// Annex G worked example on the base class: PLCopen Motion behind the standard
// handshake (S10.6). The parent Unit commands MOVE_TO exactly as it commands a
// cylinder EXTEND - it neither knows nor cares that a servo is involved (S6.1).
//
// The drive is reached ONLY through AXIS_REF and Tc2_MC2. That is what makes the
// type drive-agnostic: a Jenny Science XENAX linked as a CiA402 EtherCAT axis, a
// Beckhoff AX5000, or a simulated NC axis are the same code here. Any
// vendor-specific facility belongs in the driver layer (S10.2), never in a
// reusable CM.
//
// Like FB_SeparatorCM this type declares NO interlocks of its own (S7.2.1). Safe
// motion lives in the certified system; this module only READS its status, and
// the application supplies that status - and any station policy - through
// DeclareCondition/SetCondition. A library cannot name "STO cleared" for a
// station it has never seen.
FUNCTION_BLOCK FB_AxisCM EXTENDS FB_ControlModuleBase
VAR_INPUT
    Command : E_AxisCommand;
    ParCfg : ST_AxisParCfg;
    ParCmd : ST_AxisParCmd;
END_VAR
VAR_OUTPUT
    OutCmd : ST_AxisOutCmd;
    OutImm : ST_AxisOutImm;
    Intlk  : FB_PermIntlk;
END_VAR
VAR CONSTANT
    // §3.8b - the layout version of this module's StationCfg. It belongs with
    // the type that owns the structure, not in the reason band. Bump it when a
    // member is added or its meaning changes (§13).
    AXIS_STATIONCFG_SCHEMA : UINT := 2;   // v2 added JogRequiresEnable
END_VAR
VAR PERSISTENT
    // §3.8b - the retained image. PERSISTENT is the BACKING, not the architecture:
    // the value is registered per (Scope, WriteKey) like every other editable
    // value, so when a set store (file/JSON/XML, MES, asset system) is wired it
    // projects this through the same walk with no change here.
    // Only the VALUE is persistent - the registry's pTarget stays in ordinary
    // VAR, because a retained POINTER names nothing after a restart
    // (ST_ConfigWriteDef, TC3 §3.8b).
    _station : ST_AxisStationCfg;
END_VAR
VAR
    {attribute 'OPC.UA.DA' := '0'}
    _axis : REFERENCE TO AXIS_REF;
    {attribute 'OPC.UA.DA' := '0'}
    _recipe : I_RecipeProvider;
    {attribute 'OPC.UA.DA' := '0'}
    _power : MC_Power;
    {attribute 'OPC.UA.DA' := '0'}
    _homeFb : MC_Home;
    {attribute 'OPC.UA.DA' := '0'}
    _moveFb : MC_MoveAbsolute;
    {attribute 'OPC.UA.DA' := '0'}
    _stopFb : MC_Stop;
    {attribute 'OPC.UA.DA' := '0'}
    _resetFb : MC_Reset;
    {attribute 'OPC.UA.DA' := '0'}
    _jogFb : MC_Jog;
    _jogSeen   : BOOL;   // a held request arrived THIS scan (freshness, O10)
    _jogReqDir : INT;    // +1 / -1 / 0 as last asked
    _jogEnabled: BOOL;   // an enabling device was held when it was asked
    _jogDriving: BOOL;   // the axis is being jogged right now
    _tJogStale : TON;
    _tMove : TON;
    _homed : BOOL;
    _parCfgStaged : ST_AxisParCfg;
    _recipePrepared : BOOL;
    _appCond : ARRAY[1..PL_Fraktal.MAX_PERMINTLK_COND] OF BOOL;
END_VAR

Cyclic();

METHOD PROTECTED OnCyclic : DINT
OnCyclic := SUPER^.OnCyclic();
_M_ApplyConditions();
Intlk();
IF __ISVALIDREF(_axis) THEN                  // defensive (S5.6) [TC3]
    // Enable follows the declared conditions. Losing one drops the enable in the
    // same scan it is lost; re-enabling after it returns is a deliberate command,
    // never automatic (S9.3, S9.4).
    _power(Axis := _axis, Enable := Intlk.AllOk, Enable_Positive := Intlk.AllOk,
        Enable_Negative := Intlk.AllOk, Override := 100.0);
    OutImm.ActPos := _axis.NcToPlc.ActPos;
    OutImm.ActVelocity := _axis.NcToPlc.ActVelo;
    OutImm.DriveEnabled := _power.Status;
END_IF
_M_JogCyclic();
OutImm.TaughtPosition := _station.TaughtPosition;
OutImm.Homed := _homed;
OutCmd.Homed := _homed;
OutImm.Diagnostic := Status.Diagnostic;
END_METHOD

METHOD PRIVATE _M_ApplyConditions
VAR
    i : INT;
END_VAR
FOR i := 1 TO PL_Fraktal.MAX_PERMINTLK_COND DO
    Intlk.Cond[i] := _appCond[i];
END_FOR
END_METHOD

// Core S7.2.1 - the application names its own conditions on this module; the
// library declares none. Safe-motion status (S9.2) is read-only application
// input, so "STO cleared" is declared here by the station that can see it.
// Declared conditions start FALSE: declaring one states an intent to gate.
METHOD DeclareCondition : BOOL
VAR_INPUT
    Index : INT;
    DescriptionKey : STRING(255);
    Reason : E_Reason;
    Bypassable : BOOL;
END_VAR
IF (Index < 1) OR (Index > PL_Fraktal.MAX_PERMINTLK_COND) THEN
    DeclareCondition := FALSE;
    RETURN;
END_IF
_appCond[Index] := FALSE;
DeclareCondition := Intlk.Define(Index := Index, Description := DescriptionKey,
    Reason := Reason, Bypassable := Bypassable);
END_METHOD

// Drive a condition declared by DeclareCondition, every scan.
METHOD SetCondition : BOOL
VAR_INPUT
    Index : INT;
    Ok : BOOL;
END_VAR
IF (Index < 1) OR (Index > PL_Fraktal.MAX_PERMINTLK_COND) THEN
    SetCondition := FALSE;
    RETURN;
END_IF
_appCond[Index] := Ok;
SetCondition := TRUE;
END_METHOD

// §7.6.1 held command - JOG_POS / JOG_NEG. Called EVERY SCAN while the
// operator holds the button; silence stops the axis (see _M_JogCyclic).
//
// This method only RECORDS the request. Nothing moves from here: the decision to
// drive is taken once per scan in _M_JogCyclic, where the interlock, the enabling
// device, the freshness deadline and the command handshake are all weighed
// together. Keeping the decision in one place is what makes it reviewable.
METHOD RequestHeldCommand : BOOL
VAR_INPUT
    Value  : DINT;
    Enable : ST_ManualEnableStatus;
END_VAR
// IF rather than CASE: a CASE label must be a compile-time constant, and
// TO_DINT(enum) is a call. The intent is the same - a defined ELSE (§5.6).
IF Value = TO_DINT(E_AxisCommand.JOG_POS) THEN
    _jogReqDir :=  1;
ELSIF Value = TO_DINT(E_AxisCommand.JOG_NEG) THEN
    _jogReqDir := -1;
ELSE
    // Not a held command of this type. Refuse, and do not record it - an unknown
    // value must never leave a stale direction behind.
    RequestHeldCommand := FALSE;
    RETURN;
END_IF

_jogSeen    := TRUE;
_jogEnabled := Enable.Held;

// Refused up front, with the reason, when no safety-rated enabling device is
// permitting. The axis ALSO has to pass its interlocks in _M_JogCyclic - this is
// an additional requirement, never a way around them (§9).
//
// StationCfg.JogRequiresEnable is what an installation WITHOUT an enabling
// device declares (§3.8a). It relaxes exactly this one requirement: the
// interlocks, the freshness deadline and the command handshake are untouched,
// so a station that declares it still cannot jog through a dropped interlock
// or on a stale request.
IF _station.JogRequiresEnable AND NOT Enable.Held THEN
    OutImm.JogStopReason := PL_ModuleReasons.AXIS_JOG_NOT_ENABLED;
    RequestHeldCommand := FALSE;
    RETURN;
END_IF
RequestHeldCommand := TRUE;
END_METHOD

// The one place a jog is allowed to start, continue, or stop. Runs every scan
// from OnCyclic, whether or not anybody asked - because "nobody asked" is
// precisely the condition that has to stop the axis.
METHOD PRIVATE _M_JogCyclic
VAR
    drive : BOOL;
END_VAR
// Freshness (O10). The timer accumulates while no request arrives, so a caller
// that goes quiet - operator released, HMI closed, network stalled with the
// button still down - stops the axis after JogTimeout. A few scans of jitter are
// tolerated; a dead transport is not.
_tJogStale(IN := NOT _jogSeen, PT := ParCfg.JogTimeout);

// Every gate that must hold for the axis to move by hand, in one expression so
// there is one place to review. Interlocks are NOT bypassed for teaching: the
// station is expected to have wired its guard condition so the safety system's
// teach grant satisfies it, and if it has not, the axis simply does not jog
// (§7.2.1, fail-closed).
drive := (_jogReqDir <> 0)
    AND NOT _tJogStale.Q
    AND (_jogEnabled OR NOT _station.JogRequiresEnable)
    AND Intlk.AllOk
    AND NOT Busy                        // a commanded move owns the axis (§6.1)
    AND __ISVALIDREF(_axis);

// Say why it stopped, once, on the transition. Published status, not an alarm.
IF _jogDriving AND NOT drive THEN
    // The PLC genuinely cannot tell "operator let go" from "link died" - both
    // are simply the request no longer arriving - so it reports what it knows
    // rather than inventing a distinction. The HMI CAN tell, because it knows
    // whether it is still sending, and surfaces the difference there.
    IF _tJogStale.Q THEN
        OutImm.JogStopReason := PL_ModuleReasons.AXIS_JOG_RELEASED;
    ELSIF NOT _jogEnabled AND _station.JogRequiresEnable THEN
        OutImm.JogStopReason := PL_ModuleReasons.AXIS_JOG_NOT_ENABLED;
    ELSIF NOT Intlk.AllOk THEN
        OutImm.JogStopReason := TO_DINT(E_Reason.INTERLOCK_DROPPED);
    ELSE
        OutImm.JogStopReason := PL_ModuleReasons.AXIS_JOG_RELEASED;
    END_IF
    _jogReqDir := 0;
END_IF

IF __ISVALIDREF(_axis) THEN
    _jogFb(Axis := _axis,
           JogForward   := drive AND (_jogReqDir > 0),
           JogBackwards  := drive AND (_jogReqDir < 0),
           Mode         := MC_JOGMODE_CONTINOUS,
           Velocity     := ParCfg.JogVelocity,
           Acceleration := ParCfg.JogAcceleration,
           Deceleration := ParCfg.Deceleration);
END_IF

_jogDriving    := drive;
OutImm.Jogging := drive;
_jogSeen       := FALSE;   // consumed: the caller must ask again next scan
END_METHOD

METHOD Setup : BOOL
VAR_INPUT
    Name    : STRING(80);
    AxisRef : REFERENCE TO AXIS_REF;
    Recipe  : I_RecipeProvider;
END_VAR
VAR
    InitialModel : ST_ModelId;
END_VAR
_M_SetName(Name);
_M_SetPresentation(DisplayNameKey := 'std.moduleType.axis.name', DescriptionKey := 'std.moduleType.axis.description', TypeKey := 'std.moduleType.axis');
_axis REF= AxisRef;                      // [TC3] TC3 S3.11
_recipe := Recipe;
// No Intlk.Define here: safe-motion status and station policy are the
// application's to name (S7.2.1).
_M_PublishCommand(Value := TO_DINT(E_AxisCommand.HOME), Label := 'std.command.home');
_M_PublishCommand(Value := TO_DINT(E_AxisCommand.MOVE_TO), Label := 'std.command.moveTo');
_M_PublishHeldCommand(Value := TO_DINT(E_AxisCommand.JOG_POS), Label := 'std.command.jogPositive');
_M_PublishHeldCommand(Value := TO_DINT(E_AxisCommand.JOG_NEG), Label := 'std.command.jogNegative');
Setup := PrepareRecipe(Model := InitialModel);
IF Setup THEN CommitRecipe(); END_IF

// §3.8b restore, in one call. The rule - version 0 is a first boot that lost
// nothing, any other unrecognized version means a real image was rejected and
// is annunciated with this module's own path - is written ONCE in
// FB_ModuleBase, because every module type with a StationCfg needs exactly it
// (§1.1 O1). This type supplies only the part that is genuinely its own: what
// its declared defaults are.
//
// The CONSEQUENCE of a loss is the deployment's, not this module's: the root
// applies E_ConfigRestorePolicy. Faulting the axis here, as this used to,
// forced BLOCK_UNTIL_ACKNOWLEDGED on every station that ever used an axis.
IF NOT M_RestoreStationCfg(pVersion := ADR(_station.SchemaVersion),
        SchemaVersion := AXIS_STATIONCFG_SCHEMA) THEN
    _station.TaughtPosition := 0.0;          // this type's declared default
    // The default is the SAFE reading: an axis that lost its configuration
    // requires an enabling device again, rather than inheriting a bench's
    // relaxation into a machine that never declared one.
    _station.JogRequiresEnable := TRUE;
END_IF

// §3.8a - the taught position is an ordinary editable value: typeable by an
// engineer who knows the number, and validated against the same soft limits
// whichever way it arrives.
Setup := M_RegisterConfigNumber(Key := 'axis.taughtPosition',
    Item := 'StationCfg/TaughtPosition', LabelKey := 'std.config.axisTaughtPosition',
    Unit := E_EngUnit.MILLIMETER, Kind := E_ConfigKind.STATION_CFG, Storage := E_ConfigStorage.AS_LREAL,
    pTarget := ADR(_station.TaughtPosition), Minimum := ParCfg.SoftMin, Maximum := ParCfg.SoftMax,
    RequiresReady := FALSE) AND Setup;

// §3.8c - and it can be DEMONSTRATED instead of typed: jog the axis to the
// position, then capture. The source is OutImm.ActPos, which this module already
// publishes, so the operator sees the number before storing it (§3.8c(b)).
Setup := M_RegisterCapture(WriteKey := 'axis.taughtPosition',
    pSource := ADR(OutImm.ActPos), SourceStorage := E_ConfigStorage.AS_LREAL) AND Setup;

// §3.8a - published as an editable capability so "does this installation have
// an enabling device?" is visible, audited and carried in a station parameter
// set, instead of being a silent assumption nobody can see.
Setup := M_RegisterConfigFlag(Key := 'axis.jogRequiresEnable',
    Item := 'StationCfg/JogRequiresEnable',
    LabelKey := 'std.config.axisJogRequiresEnable',
    Kind := E_ConfigKind.STATION_CFG, pTarget := ADR(_station.JogRequiresEnable),
    RequiresReady := TRUE) AND Setup;
END_METHOD

// §3.8a/§G.4a - declare whether this INSTALLATION has a safety-rated enabling
// device for manual motion. Called by the composition root; it also stamps the
// schema version forward, so a call made before Setup survives the restore
// (a matching version is restored as-is rather than defaulted).
//
// FALSE relaxes exactly one requirement - the enabling device - and nothing
// else: interlocks, the freshness deadline and the command handshake all still
// apply, and jog still refuses a stale request. A station that declares FALSE
// should declare a §7.5 engineering gate with it, so the machine says out loud
// that it is jogging without one.
METHOD SetJogRequiresEnable : BOOL
VAR_INPUT
    Required : BOOL;
END_VAR
_station.JogRequiresEnable := Required;
_station.SchemaVersion := AXIS_STATIONCFG_SCHEMA;
SetJogRequiresEnable := TRUE;
END_METHOD

// Functional stop used by an owning sequence on abort/interlock loss. This is a
// controlled MC_Stop, NOT a certified safe stop: the safety system remains
// authoritative and STO is its business, not this module's (S9).
METHOD WithdrawOutputs
IF __ISVALIDREF(_axis) THEN
    _moveFb(Axis := _axis, Execute := FALSE);
    _homeFb(Axis := _axis, Execute := FALSE);
    // A held jog is an output of this module like any other, so it is withdrawn
    // here too - otherwise an abort would stop the commanded move and leave a
    // jog running.
    _jogFb(Axis := _axis, JogForward := FALSE, JogBackwards := FALSE);
    _stopFb(Axis := _axis, Execute := TRUE, Deceleration := ParCfg.Deceleration);
END_IF
_jogReqDir  := 0;
_jogDriving := FALSE;
OutImm.Jogging := FALSE;
_tMove(IN := FALSE);
END_METHOD

METHOD PROTECTED OnAbort : DINT
OnAbort := SUPER^.OnAbort();            // base first (S3.14.2)
WithdrawOutputs();
END_METHOD

METHOD PrepareRecipe : BOOL
VAR_INPUT
    Model : ST_ModelId;
END_VAR
IF _recipe = 0 THEN
    _parCfgStaged := ParCfg;
    _recipePrepared := TRUE;
    PrepareRecipe := TRUE;
ELSIF _recipe.Load(ModelCode := Model.ModelCode, RecipeKey := 'AxisCM', pParCfg := ADR(_parCfgStaged), Size := SIZEOF(_parCfgStaged)) THEN
    _recipePrepared := TRUE;
    PrepareRecipe := TRUE;
ELSE
    _M_Fault(E_Reason.RECIPE_INVALID, 'std.error.recipeSchemaInvalid');
    _recipePrepared := FALSE;
    PrepareRecipe := FALSE;
END_IF
END_METHOD

METHOD CommitRecipe
IF _recipePrepared THEN ParCfg := _parCfgStaged; END_IF
_recipePrepared := FALSE;
END_METHOD

METHOD AbortRecipe
_recipePrepared := FALSE;
END_METHOD

// Stop the axis, THEN fault. _M_FaultN raises the reason without touching
// motion, so faulting mid-move would leave the drive commanded - the same defect
// the separator's _M_FaultClosed exists to prevent, and worse here because the
// load is moving.
METHOD PRIVATE _M_FaultStopped
VAR_INPUT
    Code : DINT;
    Text : STRING(255);
END_VAR
WithdrawOutputs();
_M_FaultN(Code := Code, Text := Text);
END_METHOD

METHOD PROTECTED _M_PublishStatus
SUPER^._M_PublishStatus();
OutImm.Diagnostic := Status.Diagnostic;
END_METHOD

METHOD PROTECTED _M_Dispatch
VAR
    dg : ST_Diagnostic;
END_VAR
IF _manualReq THEN
    _manualReq := FALSE;
    IF (_manualCmd = TO_DINT(E_AxisCommand.HOME)) OR (_manualCmd = TO_DINT(E_AxisCommand.MOVE_TO)) THEN
        Command := _manualCmd;
    ELSE
        _M_Fault(E_Reason.UNSUPPORTED_COMMAND, 'std.error.unsupportedAxisCommand');
        RETURN;
    END_IF
END_IF
IF (Command <> E_AxisCommand.HOME) AND (Command <> E_AxisCommand.MOVE_TO) THEN
    _M_Fault(E_Reason.UNSUPPORTED_COMMAND, 'std.error.unsupportedAxisCommand');
    RETURN;
END_IF
IF Command = E_AxisCommand.HOME THEN
    _M_TagCommand(Id := 1, Label := 'std.command.home');          // S8.11.4(a)
ELSE
    _M_TagCommand(Id := 2, Label := 'std.command.moveTo');
END_IF
_M_ApplyConditions();
Intlk();
IF NOT Intlk.AllOk THEN
    // HELD, not a fault (S6.1). Losing a declared condition mid-move is expected
    // - an operator releasing an enable is the designed way to stop. The axis is
    // brought to a controlled stop by the same permit that gates the enable, and
    // the move resumes from step 10 with a full MoveTimeout window so a hold
    // cannot silently consume travel time the axis was not moving for.
    WithdrawOutputs();
    dg := Intlk.Diagnostic;
    dg.SourcePath := _name;                          // owner sets the path (S7.2)
    _M_HoldDiag(Diag := dg);
    _step := 10;
    RETURN;
END_IF
IF Command = E_AxisCommand.HOME THEN
    _M_Home();
ELSE
    _M_MoveTo();
END_IF
END_METHOD

METHOD PRIVATE _M_Home
IF NOT __ISVALIDREF(_axis) THEN
    _M_FaultN(Code := PL_ModuleReasons.AXIS_DRIVE_FAULT, Text := 'std.error.axisNotBound');
    RETURN;
END_IF
CASE _step OF
    10:
        OutCmd.InPosition := FALSE;
        _homed := FALSE;                       // homing invalidates any previous datum
        _homeFb(Axis := _axis, Execute := FALSE);
        _tMove(IN := FALSE);
        _step := 20;
    20:
        _homeFb(Axis := _axis, Execute := TRUE, Position := 0.0, HomingMode := MC_DefaultHoming);
        _tMove(IN := TRUE, PT := ParCfg.HomeTimeout);
        IF _homeFb.Done THEN
            _homeFb(Axis := _axis, Execute := FALSE);
            _tMove(IN := FALSE);
            _homed := TRUE;
            _M_Complete();
        ELSIF _homeFb.Error THEN
            _M_FaultStopped(Code := PL_ModuleReasons.AXIS_DRIVE_FAULT, Text := 'std.error.axisDriveFault');
        ELSIF _homeFb.CommandAborted THEN
            // CommandAborted means another motion command took the axis, which is
            // an abort and not a defect - route it through the base's own abort
            // path rather than inventing a fault for it.
            AbortCommand();
        ELSIF _tMove.Q THEN
            _M_FaultStopped(Code := PL_ModuleReasons.AXIS_MOVE_TIMEOUT, Text := 'std.error.axisMoveTimeout');
        END_IF
ELSE
    _M_Fault(E_Reason.STEP_STALLED, 'std.error.undefinedStep');    // defined ELSE (S5.6)
END_CASE
END_METHOD

METHOD PRIVATE _M_MoveTo
// Validate the REQUEST before the STATE, and both before commanding motion
// (S5.6). Annex G checked homed-first; range-first is used here because a target
// outside the soft limits is malformed regardless of whether the axis is homed,
// and reporting "not homed" for an impossible target sends the operator to the
// wrong problem. It also makes both rejections provable without a licensed NC
// axis, since neither issues an MC_* call.
IF (ParCmd.Target < ParCfg.SoftMin) OR (ParCmd.Target > ParCfg.SoftMax) THEN
    _M_FaultN(Code := PL_ModuleReasons.AXIS_TARGET_OOR, Text := 'std.error.axisTargetOutOfRange');
    RETURN;
END_IF
IF NOT _homed THEN
    _M_FaultN(Code := PL_ModuleReasons.AXIS_NOT_HOMED, Text := 'std.error.axisNotHomed');
    RETURN;
END_IF
IF NOT __ISVALIDREF(_axis) THEN
    _M_FaultN(Code := PL_ModuleReasons.AXIS_DRIVE_FAULT, Text := 'std.error.axisNotBound');
    RETURN;
END_IF
CASE _step OF
    10:
        OutCmd.InPosition := FALSE;
        _moveFb(Axis := _axis, Execute := FALSE);
        _tMove(IN := FALSE);
        _step := 20;
    20:
        // MC_MoveAbsolute's Busy/Done/Error/CommandAborted map one-to-one onto
        // the CM handshake, which is what lets a parent Unit command MOVE_TO
        // exactly as it commands a cylinder EXTEND (S6.1).
        _moveFb(Axis := _axis, Execute := TRUE, Position := ParCmd.Target,
            Velocity := ParCfg.Velocity, Acceleration := ParCfg.Acceleration,
            Deceleration := ParCfg.Deceleration);
        _tMove(IN := TRUE, PT := ParCfg.MoveTimeout);
        IF _moveFb.Done THEN
            _moveFb(Axis := _axis, Execute := FALSE);
            _tMove(IN := FALSE);
            OutCmd.InPosition := TRUE;
            _M_Complete();
        ELSIF _moveFb.Error THEN
            _M_FaultStopped(Code := PL_ModuleReasons.AXIS_DRIVE_FAULT, Text := 'std.error.axisDriveFault');
        ELSIF _moveFb.CommandAborted THEN
            // CommandAborted means another motion command took the axis, which is
            // an abort and not a defect - route it through the base's own abort
            // path rather than inventing a fault for it.
            AbortCommand();
        ELSIF _tMove.Q THEN
            _M_FaultStopped(Code := PL_ModuleReasons.AXIS_MOVE_TIMEOUT, Text := 'std.error.axisMoveTimeout');
        END_IF
ELSE
    _M_Fault(E_Reason.STEP_STALLED, 'std.error.undefinedStep');
END_CASE
END_METHOD

END_FUNCTION_BLOCK

(* stored: Version 1.1.0.1, ProductVersion 3.1.4024.12
   POU FB_AxisCM: Id {67f6d9e3-e1d3-4e52-8c0e-a2b82552da28}, SpecialFunc None
   Method OnCyclic: Id {2294d08b-7382-44fe-95ee-1e560113af12}
   Method _M_ApplyConditions: Id {7c42158c-5f9f-4b6d-9d24-a2ceb651080e}
   Method DeclareCondition: Id {523d6056-ce78-4c1f-bac4-a4fb8c004e4b}
   Method SetCondition: Id {4bd35f8a-650f-45f8-b8f5-2559d8a0b7f9}
   Method RequestHeldCommand: Id {8b520989-3ece-43bf-8be8-d0b6fb508907}
   Method _M_JogCyclic: Id {8ac1844d-58f5-43a2-9230-a4104ef57973}
   Method Setup: Id {b344bdf9-c716-4e60-b22e-283b03a3f9b4}
   Method SetJogRequiresEnable: Id {6e2f90a4-53d1-4c78-b0a6-9d3417e285fb}
   Method WithdrawOutputs: Id {7048fa32-48b6-4490-a0f4-1a93a00524fb}
   Method OnAbort: Id {e9fcd5a6-e437-44a3-9c68-4beda7d104fb}
   Method PrepareRecipe: Id {06ac63ce-5078-4aaa-8399-955a5acacc2e}
   Method CommitRecipe: Id {4c30e8ed-295f-4209-bc77-bb72e178711b}
   Method AbortRecipe: Id {8126c3c3-0571-4320-8290-d4bd17d0b684}
   Method _M_FaultStopped: Id {64e28450-10e9-4a76-9816-bbd8fc289187}
   Method _M_PublishStatus: Id {e9a88f13-6d14-431a-a265-e23cd64cdaeb}
   Method _M_Dispatch: Id {fd1c6a2e-126f-4404-a707-69fd01270561}
   Method _M_Home: Id {186051b1-bda7-4b8e-9bd9-ab8bf047605f}
   Method _M_MoveTo: Id {95306de5-b879-4b0c-a486-0cd807e9bc83} *)
